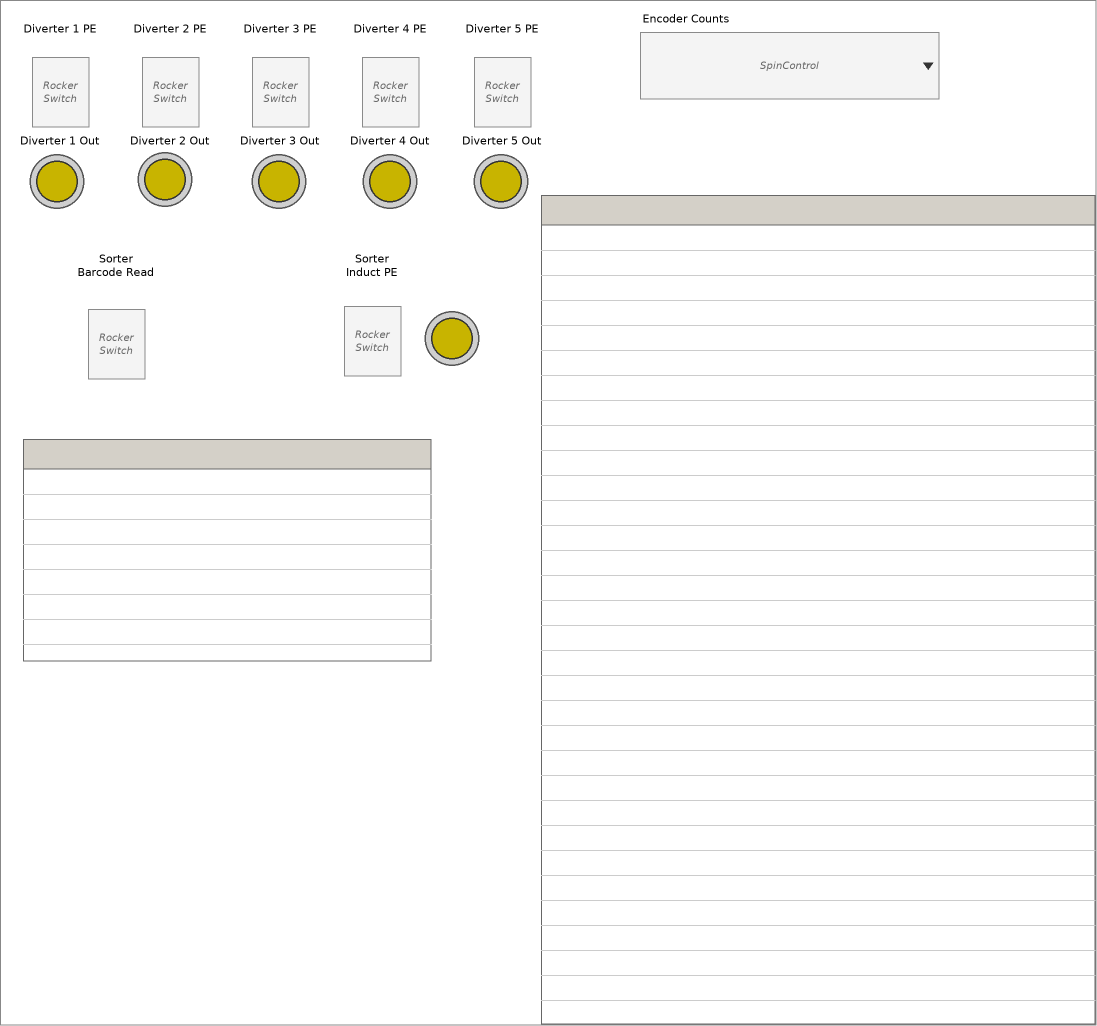
VISUALIZATION DiverterTest  // 1097x1026
    RockerSwitch (32,57 57x70), variable: Diverts[1].JamPE, behaviour: TOGGLE, style: Switch-RockerSwitch-Blue
    Label (9,10 102x38), "Diverter 1 PE"
    RockerSwitch (142,57 57x70), variable: Diverts[2].JamPE, behaviour: TOGGLE, style: Switch-RockerSwitch-Blue
    Label (119,10 102x38), "Diverter 2 PE"
    RockerSwitch (252,57 57x70), variable: Diverts[3].JamPE, behaviour: TOGGLE, style: Switch-RockerSwitch-Blue
    Label (229,10 102x38), "Diverter 3 PE"
    RockerSwitch (362,57 57x70), variable: Diverts[4].JamPE, behaviour: TOGGLE, style: Switch-RockerSwitch-Blue
    Label (339,10 102x38), "Diverter 4 PE"
    RockerSwitch (474,57 57x70), variable: Diverts[5].JamPE, behaviour: TOGGLE, style: Switch-RockerSwitch-Blue
    Label (451,10 102x38), "Diverter 5 PE"
    RockerSwitch (88,309 57x70), variable: BarcodeRead, behaviour: TOGGLE, style: Switch-RockerSwitch-Blue
    Label (65,231 102x69), "Sorter Barcode Read"
    SpinControl (640,32 299x67), variable: MAIN.Sorter1.CurrentRead
    Lamp1 (25,150 64x63), variable: Diverts[1].Output1, style: Lamp-Lamp1-Yellow
    Lamp1 (133,148 64x63), variable: Diverts[2].Output1, style: Lamp-Lamp1-Yellow
    Lamp1 (247,150 64x63), variable: Diverts[3].Output1, style: Lamp-Lamp1-Yellow
    Lamp1 (358,150 64x63), variable: Diverts[4].Output1, style: Lamp-Lamp1-Yellow
    Lamp1 (469,150 64x63), variable: Diverts[5].Output1, style: Lamp-Lamp1-Yellow
    RockerSwitch (344,306 57x70), variable: SorterinductPE, behaviour: TOGGLE, style: Switch-RockerSwitch-Blue
    Label (321,231 102x69), "Sorter Induct PE"
    Lamp1 (420,307 64x63), variable: SorterinductPE, style: Lamp-Lamp1-Yellow
    Table (541,195 554x829), data array: MAIN.aSorterItems
        p3854506369: MAIN.aSorterItems[INDEX].ID
        p2232123230: MAIN.SorterItems[INDEX].ID
        p511219082: MAIN.SorterItems[INDEX].UniqueID
        p1892666644: MAIN.aSorterItems[INDEX].UniqueID
        p1755163831: MAIN.SorterItems[INDEX].Destination
        p338671338: MAIN.aSorterItems[INDEX].Destination
        p4092479075: MAIN.SorterItems[INDEX].Status
        p2170511999: MAIN.aSorterItems[INDEX].Status
        p3723444502: MAIN.aSorterItems[INDEX].CapturedInMetrics
        p2237128397: MAIN.SorterItems[INDEX].CapturedInMetrics
    Table (23,439 408x222), data array: ArrivalOut
        p1755163831: ArrivalOut[INDEX].Destination
        p4092479075: ArrivalOut[INDEX].Status
        p2232123230: ArrivalOut[INDEX].UniqueID
        p511219082: ArrivalOut[INDEX].ID
    Label (9,122 102x38), "Diverter 1 Out"
    Label (119,122 102x38), "Diverter 2 Out"
    Label (229,122 102x38), "Diverter 3 Out"
    Label (339,122 102x38), "Diverter 4 Out"
    Label (451,122 102x38), "Diverter 5 Out"
    Label (635,0 102x38), "Encoder Counts"
END_VISUALIZATION

(* stored: Version 1.1.0.1, ProductVersion 3.1.4024.4
   Visu DiverterTest: Id {45e687eb-88c1-40e7-bcf9-5ec7b05235a8} *)
